(* IEC 61131-3 sources: Industry-PLC-LLM/data/PLCBEAD_repo/PLCBEAD_PLCEmbed-main/PLC-BEAD/Source/GEB/building_SDD, 1 file *)

(* ---- SDD.ST ---- *)
FUNCTION SDD:REAL

	VAR_INPUT
		T :	REAL;
		ICE :	BOOL;
	END_VAR

	IF ice THEN
		SDD := 611.153 * EXP(22.4433 * T / (272.186 + T));
	ELSE
		SDD := 611.213 * EXP(17.5043 * T / (241.2 + T));
	END_IF;

END_FUNCTION

PROGRAM program0
  VAR
    T :	REAL;
	ICE :	BOOL;
    CEIL5_OUT : REAL;
  END_VAR

  CEIL5_OUT := SDD(T, ICE);
END_PROGRAM
